// TIA Portal V21 export
TYPE "Rcp_Blower&Rinser"
   STRUCT
      AltezzaCarosello : Real;
      Abilitazione1Trattamento : Bool;
   END_STRUCT;
END_TYPE
